TYPE ST_ComponentVisu :
STRUCT
	sName				: STRING;
	bError				: BOOL;
	bRunning			: BOOL;
	bReset				: BOOL;
	bEnable				: BOOL;
	bAccessPermit		: BOOL;
	eState				: E_ComponentState;
	colBackground		: DWORD;
END_STRUCT
END_TYPE

(* stored: Version 1.1.0.1
   DUT ST_ComponentVisu: Id {6c5249ce-4a17-4379-aa00-249f9406ce52} *)
